# B&R Automation Studio project ServoMgr
Automation Studio 4.11.2.75; technology packages: Acp10Arnc0 5.12.2

## Configuration ARM

CPU X20CP0410, AutomationRuntime B4.92, Build 6.3.0, Vc V4.72.5

### Task classes (Cpu.sw)
```
Cyclic#1:
  FirstInitP <- Infrastructure.FirstInitProg.prg
Cyclic#3:
  ServoMgr <- Servo.ServoMgr.prg
Cyclic#4:
  MachinePro <- MachineControl.MachineProg.prg
Cyclic#8:
  ErrorProg <- Diagnostics.ErrorProg.prg
  MachineHMI <- MachineControl.MachineHMI.prg
DataObjects: Acp10sys
Binaries: udbdef, FWRules, TCData, acp10cfg, Acp10map, iomap, asfw, Role, sysconf, arconfig, ashwd, User, ashwac
Libraries: operator, runtime, astime, AsIecCon, sys_lib, AsBrStr, ArEventLog, AsBrWStr, Acp10_MC, Acp10man, Acp10par, NcGlobal, brsystem, standard, FileIO, AsArLog, asstring, AxisLib, persist, csvfilelib, fiowrap, stringext, hmitools, ringbuflib, logthat, piper, errorlib, vartools, powerlnk, axiserrlib
```

## Configuration Config1

CPU 5PC900.TS17-00, AutomationRuntime E4.92, Build 4.1.2, Safety 0.0, Vc V4.72.5

### Task classes (Cpu.sw)
```
Cyclic#1:
  FirstInitP <- Infrastructure.FirstInitProg.prg
Cyclic#3:
  ServoMgr <- Servo.ServoMgr.prg
Cyclic#4:
  cPiperModu <- MachineControl.cPiperModuleTemplate.prg
  MachineHMI <- MachineControl.MachineHMI.prg
  MachinePro <- MachineControl.MachineProg.prg
  PiperModul <- MachineControl.PiperModuleTemplate.prg
  ErrorProg <- Diagnostics.ErrorProg.prg
DataObjects: Acp10sys
Binaries: udbdef, FWRules, TCData, acp10cfg, Acp10map, iomap, asfw, Role, sysconf, arconfig, ashwd, User, ashwac
Libraries: operator, sys_lib, AsBrStr, runtime, ArEventLog, astime, AsBrWStr, brsystem, Acp10man, Acp10par, NcGlobal, standard, FileIO, AsArLog, AxisLib, asstring, Acp10_MC, piper, stringext, logthat, AxisErrLib, errorlib, hmitools, ringbuflib, csvfilelib, fiowrap, persist, vartools, powerlnk, asieccon
```

## Configuration Intel

CPU 5PC900.TS17-00, AutomationRuntime B4.92, Build 4.1.2, Safety 0.0, Vc V4.72.5

### Task classes (Cpu.sw)
```
Cyclic#1:
  FirstInitP <- Infrastructure.FirstInitProg.prg
Cyclic#3:
  ServoMgr <- Servo.ServoMgr.prg
Cyclic#4:
  MachinePro <- MachineControl.MachineProg.prg
Cyclic#8:
  ErrorProg <- Diagnostics.ErrorProg.prg
  MachineHMI <- MachineControl.MachineHMI.prg
DataObjects: Acp10sys
Binaries: udbdef, FWRules, TCData, acp10cfg, Acp10map, iomap, asfw, Role, sysconf, arconfig, ashwd, User, ashwac
Libraries: operator, sys_lib, AsBrStr, runtime, ArEventLog, astime, AsBrWStr, brsystem, Acp10man, Acp10par, NcGlobal, standard, FileIO, AsArLog, AxisLib, asstring, Acp10_MC, piper, persist, csvfilelib, fiowrap, vartools, errorlib, hmitools, ringbuflib, logthat, stringext, powerlnk, axiserrlib, asieccon
```

### Acp10cfg.ncc - 5PC900_TS17_00/Motion/Acp10cfg.ncc
```
NcConfiguration (Version=5.23.1, NcSwId=Acp10)
  ACP10CF1_typ:
    cnt_nettrc_rec_drive = 150
    bufsize_trace_upload = 1200
    tc_nc_man_task = Cyclic #1
    glob_pv_as_ncobject = Yes
    ncsys_dl_broadcast = Yes
    ncsys_dl_acp_reset = Yes
    safemc_log_err_to_ax = Yes
    network_init:
      ncsw_init_execute = Yes
      automatic_execute = No
      node_nr_warning = Yes
      net_err_before_ncact = Yes
    nettrc:
      enter_parsecrec = Yes
      enter_ncaction = Yes
      save_ring_startidx = No
    cam_prof_download:
      cam_dat_dl_parallel = No
      tc_cam_dl_parallel = Task class for NC Manager task
```

## Logical view

Binary libraries used (declarations not repeated): operator, runtime, astime, AsIecCon, sys_lib, AsBrStr, ArEventLog, AsBrWStr, Acp10_MC 5.17.1, Acp10man 5.17.1, Acp10par, NcGlobal, brsystem, standard, FileIO, AsArLog, asstring, AxisLib, piper, stringext, logthat 0.05.1, axiserrlib 0.00.5, errorlib 0.23.3, hmitools, ringbuflib, csvfilelib 1.02.2, fiowrap 0.09.1, persist 0.00.7, vartools 0.11.3


### Program Logical/Infrastructure/FirstInitProg (IEC)

#### Init.st - Init code
```iecst
(*******************************************************************
* COPYRIGHT --
********************************************************************
* PROGRAM: FirstInitProg
* File: FirstInitProgInit.c
* Author: ScismD
* Created: January 07, 2014
********************************************************************
* Implementation OF PROGRAM FirstInitProg
*******************************************************************)

PROGRAM _INIT
	// Check for simulation
	// This is a DevLink using a Windows share which is not supported by ARsim
	// We use this instead of Diag function to support older CPU's
	simCheckDevLink.enable := TRUE;
	simCheckDevLink.pDevice := ADR('SimCheck');
	simCheckDevLink.pParam := ADR('/SIP=127.0.0.1 /PROTOCOL=cifs /SHARE=testfolder /USER=max /PASSWORD=passw');

	simCheckDevLink();

	IF (simCheckDevLink.status = ERR_NOTIMPLEMENTED) THEN
		gSimulation := TRUE;
	END_IF

	// Initialize User Loggers
	createLogInit('Errors', 1000000, arEVENTLOG_PERSISTENCE_VOLATILE);
	createLogInit('Files', 1000000, arEVENTLOG_PERSISTENCE_VOLATILE);
	createLogInit('Application', 1000000, arEVENTLOG_PERSISTENCE_VOLATILE);

	// Initialize error collector
	ErrorCollectorFn_Init(gErrorCollector);

	// Link file devices
	//-------------------------------------------------------

	// This is NOT done in the CPU configuration because when using CPU simulation
	// you cannot have separate file devices for simulation mode,
	// and you cannot unlink devices that were entered in the CPU configuration

	// Set up file device names
	brsstrcpy(ADR(fileDevice[0]), ADR('CF_User'));
	brsstrcpy(ADR(fileDevice[1]), ADR('CNC_PrgDir'));
	brsstrcpy(ADR(fileDevice[2]), ADR('Recipes'));
	brsstrcpy(ADR(fileDevice[3]), ADR('permBackup'));

	// Set up file device paths
	IF (gSimulation) THEN
		brsstrcpy(ADR(directory[0]), ADR('C:\\ARSimUser\\LamResearch_MiniCell'));
		brsstrcpy(ADR(directory[1]), ADR('C:\\ARSimUser\\LamResearch_MiniCell\\CNC'));
		brsstrcpy(ADR(directory[2]), ADR('C:\\ARSimUser\\LamResearch_MiniCell\\Recipes'));
		brsstrcpy(ADR(directory[3]), ADR('C:\\ARSimUser\\LamResearch_MiniCell\\PermData'));
	ELSE
		brsstrcpy(ADR(directory[0]), ADR('F:\\'));
		brsstrcpy(ADR(directory[1]), ADR('F:\\CNC'));
		brsstrcpy(ADR(directory[2]), ADR('F:\\Recipes'));
		brsstrcpy(ADR(directory[3]), ADR('F:\\PermData'));
	END_IF

	// Link file devices
	FOR i:=0 TO MAI_FILEDEVICES BY 1 DO

		brsstrcpy(ADR(parameters[i]), ADR('/DEVICE='));
		stringlcat(ADR(parameters[i]), ADR(directory[i]), SIZEOF(parameters[i]));

		fileDeviceDevLink[i].enable := TRUE;
		fileDeviceDevLink[i].pDevice := ADR(fileDevice[i]);
		fileDeviceDevLink[i].pParam := ADR(parameters[i]);

		fileDeviceDevLink[i]();

		IF (fileDeviceDevLink[i].status <> 0) THEN
			errcolAddError(ADR('File Devices'), ADR('Error linking file device'), fileDeviceDevLink[i].status, 0, gErrorCollector);
		END_IF

	END_FOR

	// Initialize Persisters
	//-------------------------------------------------------

	// Working variables

	// Machine configuration
	foundVars := varGetVariableList(ADR('Configuration'), ADR(gPersister[PERM_CONFIGURATION].IN.WorkingVariableList));

	// Home data
	brsstrcpy(ADR(gPersister[PERM_HOME_DATA].IN.WorkingVariableList[0]),ADR('gEndlessPosition'));

	// Axis pars
	// Verify that NUM_MOTOR is defined by ServoControl if error occurs here
	FOR i := 0 TO MAI_MOTOR BY 1 DO
		brsitoa(i, ADR(indexString));
		brsstrcpy(ADR(axisString), ADR('gMotorBasic'));
		appendArrayIndex(i, ADR(axisString));
		stringlcat(ADR(axisString),ADR('.IN.PAR'),SIZEOF(axisString));

		IF (i <= PERSIST_MAI_VARLIST) THEN
			brsstrcpy(ADR(gPersister[PERM_AXIS_PARS].IN.WorkingVariableList[i]), ADR(axisString));
		ELSE
			errcolAddError(ADR('Perm Data'), ADR('Too many axes for one persister.'), 0, 0, gErrorCollector);
			EXIT;
		END_IF

	END_FOR

	// Axis cfg
	// Verify that NUM_MOTOR is defined by ServoControl if error occurs here
	FOR i := 0 TO MAI_MOTOR BY 1 DO
		brsitoa(i, ADR(indexString));
		brsstrcpy(ADR(axisString), ADR('gMotorBasic'));
		appendArrayIndex(i, ADR(axisString));
		stringlcat(ADR(axisString),ADR('.IN.CFG'),SIZEOF(axisString));

		IF (i <= PERSIST_MAI_VARLIST) THEN
			brsstrcpy(ADR(gPersister[PERM_AXIS_CFG].IN.WorkingVariableList[i]), ADR(axisString));
		ELSE
			errcolAddError(ADR('Perm Data'), ADR('Too many axes for one persister.'), 0, 0, gErrorCollector);
			EXIT;
		END_IF

	END_FOR

	// Permanent variables
	gPersister[PERM_CONFIGURATION].IN.pPersistentVariable := ADR(gPermConfiguration);
	gPersister[PERM_CONFIGURATION].IN.sizeofPersistentVariable := SIZEOF(gPermConfiguration);

	gPersister[PERM_HOME_DATA].IN.pPersistentVariable := ADR(gPermHomeData);
	gPersister[PERM_HOME_DATA].IN.sizeofPersistentVariable := SIZEOF(gPermHomeData);

	gPersister[PERM_AXIS_PARS].IN.pPersistentVariable := ADR(gPermAxisPars);
	gPersister[PERM_AXIS_PARS].IN.sizeofPersistentVariable := SIZEOF(gPermAxisPars);

	gPersister[PERM_AXIS_CFG].IN.pPersistentVariable := ADR(gPermAxisCfgs);
	gPersister[PERM_AXIS_CFG].IN.sizeofPersistentVariable := SIZEOF(gPermAxisCfgs);

	// DataValid and PersistFn_Init()
	FOR i := 0 TO MAI_PERSISTERS BY 1 DO
		gPersister[i].IN.pDataValid := ADR(gDataValid[i]);
		PersistFn_Init(gPersister[i]);
		IF (gPersister[i].OUT.STAT.Error) THEN
			errcolAddError(ADR('Perm Data'), ADR(gPersister[i].OUT.STAT.ErrorString), gPersister[i].OUT.STAT.ErrorID, 0, gErrorCollector);
		END_IF
	END_FOR

	// Initialize persister CSV backups
	errcolAddSourceByName(ADR('Machine configuration backup'), ADR('gPermBackup[0]'), gErrorCollector);
	errcolAddSourceByName(ADR('Home data backup'), ADR('gPermBackup[1]'), gErrorCollector);
	errcolAddSourceByName(ADR('Axis pars backup'), ADR('gPermBackup[2]'), gErrorCollector);
	errcolAddSourceByName(ADR('Axis cfg backup'), ADR('gPermBackup[3]'), gErrorCollector);

	brsstrcpy(ADR(gPermBackup[PERM_CONFIGURATION].IN.PAR.FileName), ADR('configuration.csv'));
	brsstrcpy(ADR(gPermBackup[PERM_HOME_DATA].IN.PAR.FileName), ADR('homeData.csv'));
	brsstrcpy(ADR(gPermBackup[PERM_AXIS_PARS].IN.PAR.FileName), ADR('axisPars.csv'));
	brsstrcpy(ADR(gPermBackup[PERM_AXIS_CFG].IN.PAR.FileName), ADR('axisCfg.csv'));

	FOR i := 0 TO MAI_PERSISTERS BY 1 DO

		brsstrcpy(ADR(gPermBackup[i].IN.PAR.FileDevice), ADR('permBackup'));
		brsmemcpy(ADR(gPermBackup[i].IN.PAR.VariableList), ADR(gPersister[i].IN.WorkingVariableList), SIZEOF(gPermBackup[i].IN.PAR.VariableList));

		brsstrcpy(ADR(gPermBackup[i].IN.CFG.LogFileName), ADR('.csvlogPermBackup'));
		brsitoa(i, ADR(indexString));
		brsstrcat(ADR(gPermBackup[i].IN.CFG.LogFileName), ADR(indexString));

		CSVFn_Init(gPermBackup[i]);

		IF (NOT gDataValid[i]) THEN
			CSVOpenFile_Init(gPermBackup[i]);
			IF (NOT gPermBackup[i].OUT.STAT.Error) THEN
				gDataValid[i] := TRUE;
				errcolAddError(ADR('Data restored'), ADR(gPermBackup[i].IN.PAR.FileName), 0, 0, gErrorCollector);
			END_IF
		END_IF

	END_FOR // loop through permbackup

	// Load configuration.csv every startup
	//CSVOpenFile_Init(&gPermBackup[PERM_CONFIGURATION]);

	gClearTrace := 1;

END_PROGRAM
```

#### Cyclic.st - Cyclic code
```iecst
PROGRAM _CYCLIC
	// DO NOT ADD ANY CYCLIC CODE HERE! //

END_PROGRAM
```

#### Variables.var - Local variables
```iecst
VAR CONSTANT
	NUM_FILEDEVICES : USINT := 4;
	MAI_FILEDEVICES : USINT := NUM_FILEDEVICES-1;
END_VAR
VAR
	simCheckDevLink : DevLink := (0);
	fileDeviceDevLink : ARRAY[0..MAI_FILEDEVICES] OF DevLink := [4(0)];
	fileDevice : ARRAY[0..MAI_FILEDEVICES] OF STRING[20] := [4('')];
	directory : ARRAY[0..MAI_FILEDEVICES] OF STRING[320] := [4('')];
	parameters : ARRAY[0..MAI_FILEDEVICES] OF STRING[320] := [4('')];
	i : DINT := 0;
	indexString : STRING[320] := '';
	axisString : STRING[320] := '';
	foundVars : UINT;
END_VAR
```

### Infrastructure.var
```iecst
(*Constants for number of persisters and permanent memory chunks*)
VAR CONSTANT
	NUM_PERSISTERS : USINT := 4;
	MAI_PERSISTERS : USINT := NUM_PERSISTERS-1;
END_VAR
(*Persisters to handle memory management*)
VAR
	gSimulation : BOOL;
	gPersister : ARRAY[0..MAI_PERSISTERS] OF Persistence_typ;
	gPermBackup : ARRAY[0..MAI_PERSISTERS] OF CSVFileMgr_typ;
END_VAR
VAR RETAIN
	gDataValid : ARRAY[0..MAI_PERSISTERS] OF BOOL;
END_VAR
(*Permanent memory chunks*)
VAR RETAIN
	gPermHomeData : ARRAY[0..999] OF USINT;
	gPermAxisPars : ARRAY[0..4999] OF USINT;
	gPermAxisCfgs : ARRAY[0..999] OF USINT;
	gPermConfiguration : ARRAY[0..1999] OF USINT;
END_VAR
VAR
	gClearTrace : BOOL;
END_VAR
```

### Program Logical/MachineControl/cPiperModuleTemplate (ANSIC)

#### PiperModule.var
```iecst
(********************************************************************
 * COPYRIGHT --
 ********************************************************************
 * Program: cPiperModuleTemplate
 * File: cPiperModuleTemplate.var
 * Author: dfblackburn
 * Created: April 06, 2016
 ********************************************************************
 * Local variables of program cPiperModuleTemplate
 ********************************************************************)
VAR
	ModuleInterface : Module_Interface_typ;
	Module : Piper_Module_Fub;
END_VAR
```

### MachineControl.typ
```iecst
(********************************************************************
 * COPYRIGHT -- Automation Resources Group
 ********************************************************************
 * Package: MachineControl
 * File: MachineControl.typ
 * Author: David Blackburn
 * Created: November 10, 2011
 ********************************************************************
 * Data types of package MachineControl
 ********************************************************************)

TYPE
	SUBSTATES :
		(
		SUB_STATE_INIT,
		SUB_STATE_SAFETY_RESET,
		SUB_STATE_SERVO_POWER,
		SUB_STATE_ENABLE_AXIS_ENAGAGE,
		SUB_STATE_ENABLE_PATH_SYNC,
		SUB_STATE_STARTING_SET_AXES,
		SUB_STATE_STARTING_CNC_LIMITS,
		SUB_STATE_STARTING_AXIS_LIMITS,
		SUB_STATE_STARTING_CNC_START,
		SUB_STATE_STARTING_CNC_STARTED,
		SUB_STATE_STARTING_CNC_FAILED,
		SUB_STATE_STOPPING_STOP_CNC,
		SUB_STATE_DISABLE_AXIS_ENAGAGE,
		SUB_STATE_SERVO_STOP,
		SUB_STATE_SERVO_POWER_OFF
		);
	MODE_MACHINE_ENUM :
		(
		MODE_MACHINE_AUTO,
		MODE_MACHINE_MANUAL_PROGRAM,
		MODE_MACHINE_MANUAL_JOG
		);

END_TYPE
```

- Program Logical/MachineControl/MachineHMI (IEC) (no source held here)

### Program Logical/MachineControl/MachineProg (IEC)

#### MachineProg.var - Local variables
```iecst
(********************************************************************
 * COPYRIGHT -- Automation Resources Group
 ********************************************************************
 * Program: MachineProg
 * File: MachineProg.var
 * Author: David Blackburn
 * Created: November 10, 2011
 ********************************************************************
 * Local variables of program MachineProg
 ********************************************************************)
VAR
	StatusModule : Module_Interface_typ;
	Module : REFERENCE TO Module_Interface_typ;
	TON_0 : TON;
	StateString : STRING[80];
END_VAR
VAR RETAIN
	ByPassAll : BOOL := 0;
END_VAR
```

### Package Logical/Diagnostics - Diagnostics software

### Diagnostics.var
```iecst
(********************************************************************
 * COPYRIGHT --
 ********************************************************************
 * Package: Diagnostics
 * File: Diagnostics.var
 * Author: davidblackburn
 * Created: December 20, 2013
 ********************************************************************
 * Variables of package Diagnostics
 ********************************************************************)
(*Error collector*)
VAR
	gErrorCollector : ErrorCollector_typ := (0);
	gErrorCollectorHMI : ErrorCollector_HMI_typ := (0);
END_VAR
```

- Program Logical/Diagnostics/ErrorProg (IEC) (no source held here)

Listed in the project but not available here: Logical/Global.typ, Logical/Global.var, Logical/Infrastructure/FirstInitProg/Types.typ, Logical/Infrastructure/Infrastructure.typ, Logical/MachineControl/MachineControl.var, Logical/MachineControl/MachineHMI/MachineProgCyclic.st, Logical/MachineControl/MachineHMI/MachineProgInit.st, Logical/MachineControl/MachineHMI/MachineProg.typ, Logical/MachineControl/MachineHMI/MachineProg.var, Logical/MachineControl/MachineProg/MachineProgCyclic.st, Logical/MachineControl/PiperModuleTemplate, C:/Projects/Loupe/AxisLib/src/Ar/Servo, Logical/Diagnostics/ErrorProg/ErrorProgInit.st, Logical/Diagnostics/ErrorProg/ErrorProgCyclic.st, Logical/Diagnostics/ErrorProg/ErrorProg.typ, Logical/Diagnostics/ErrorProg/ErrorProg.var, Logical/Diagnostics/ErrorProg/PiperModuleTemplate.var, Logical/Diagnostics/ErrorProg/PiperModuleInterface.st
